# EPICS autosave request: ADBruker/brukerApp/Db/BIS_settings.req
$(P)$(R)ReadSFRMTimeout
$(P)$(R)NumDarks
